FUNCTION_BLOCK Server_ALL (* Composite Function Block Type *)
  (* Standard: 61499-2 *)
  (* Version 0.0, 2018-11-07, 4DIAC-IDE, 4DIAC-Consortium *)
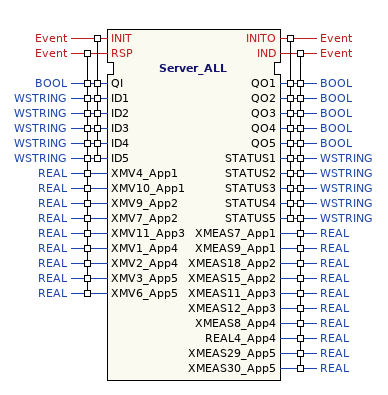
  EVENT_INPUT
    INIT WITH QI, ID1, ID2, ID4, ID5, ID3; (* Initialization Request *)
    RSP WITH QI, ID1, ID2, ID3, ID4, ID5, XMV4_App1, XMV10_App1, XMV9_App2, XMV7_App2, XMV11_App3, XMV1_App4, XMV2_App4, XMV3_App5, XMV6_App5; (* Normal Execution Request *)
  END_EVENT
  EVENT_OUTPUT
    INITO WITH QO1, QO3, QO2, QO4, QO5, STATUS1, STATUS2, STATUS3, STATUS4, STATUS5; (* Initialization Confirm *)
    IND WITH QO1, QO2, QO3, QO4, QO5, STATUS2, STATUS1, STATUS3, STATUS4, STATUS5, XMEAS7_App1, XMEAS9_App1, XMEAS18_App2, XMEAS15_App2, XMEAS11_App3, XMEAS12_App3, XMEAS8_App4, REAL4_App4, XMEAS29_App5, XMEAS30_App5; (* Execution Confirmation *)
  END_EVENT
  VAR_INPUT
    QI : BOOL; (* Input event qualifier *)
    ID1 : WSTRING;
    ID2 : WSTRING;
    ID3 : WSTRING;
    ID4 : WSTRING;
    ID5 : WSTRING;
    XMV4_App1 : REAL;
    XMV10_App1 : REAL;
    XMV9_App2 : REAL;
    XMV7_App2 : REAL;
    XMV11_App3 : REAL;
    XMV1_App4 : REAL;
    XMV2_App4 : REAL;
    XMV3_App5 : REAL;
    XMV6_App5 : REAL;
  END_VAR
  VAR_OUTPUT
    QO1 : BOOL; (* Output event qualifier *)
    QO2 : BOOL;
    QO3 : BOOL;
    QO4 : BOOL;
    QO5 : BOOL;
    STATUS1 : WSTRING;
    STATUS2 : WSTRING;
    STATUS3 : WSTRING;
    STATUS4 : WSTRING;
    STATUS5 : WSTRING;
    XMEAS7_App1 : REAL;
    XMEAS9_App1 : REAL;
    XMEAS18_App2 : REAL;
    XMEAS15_App2 : REAL;
    XMEAS11_App3 : REAL;
    XMEAS12_App3 : REAL;
    XMEAS8_App4 : REAL;
    REAL4_App4 : REAL;
    XMEAS29_App5 : REAL;
    XMEAS30_App5 : REAL;
  END_VAR
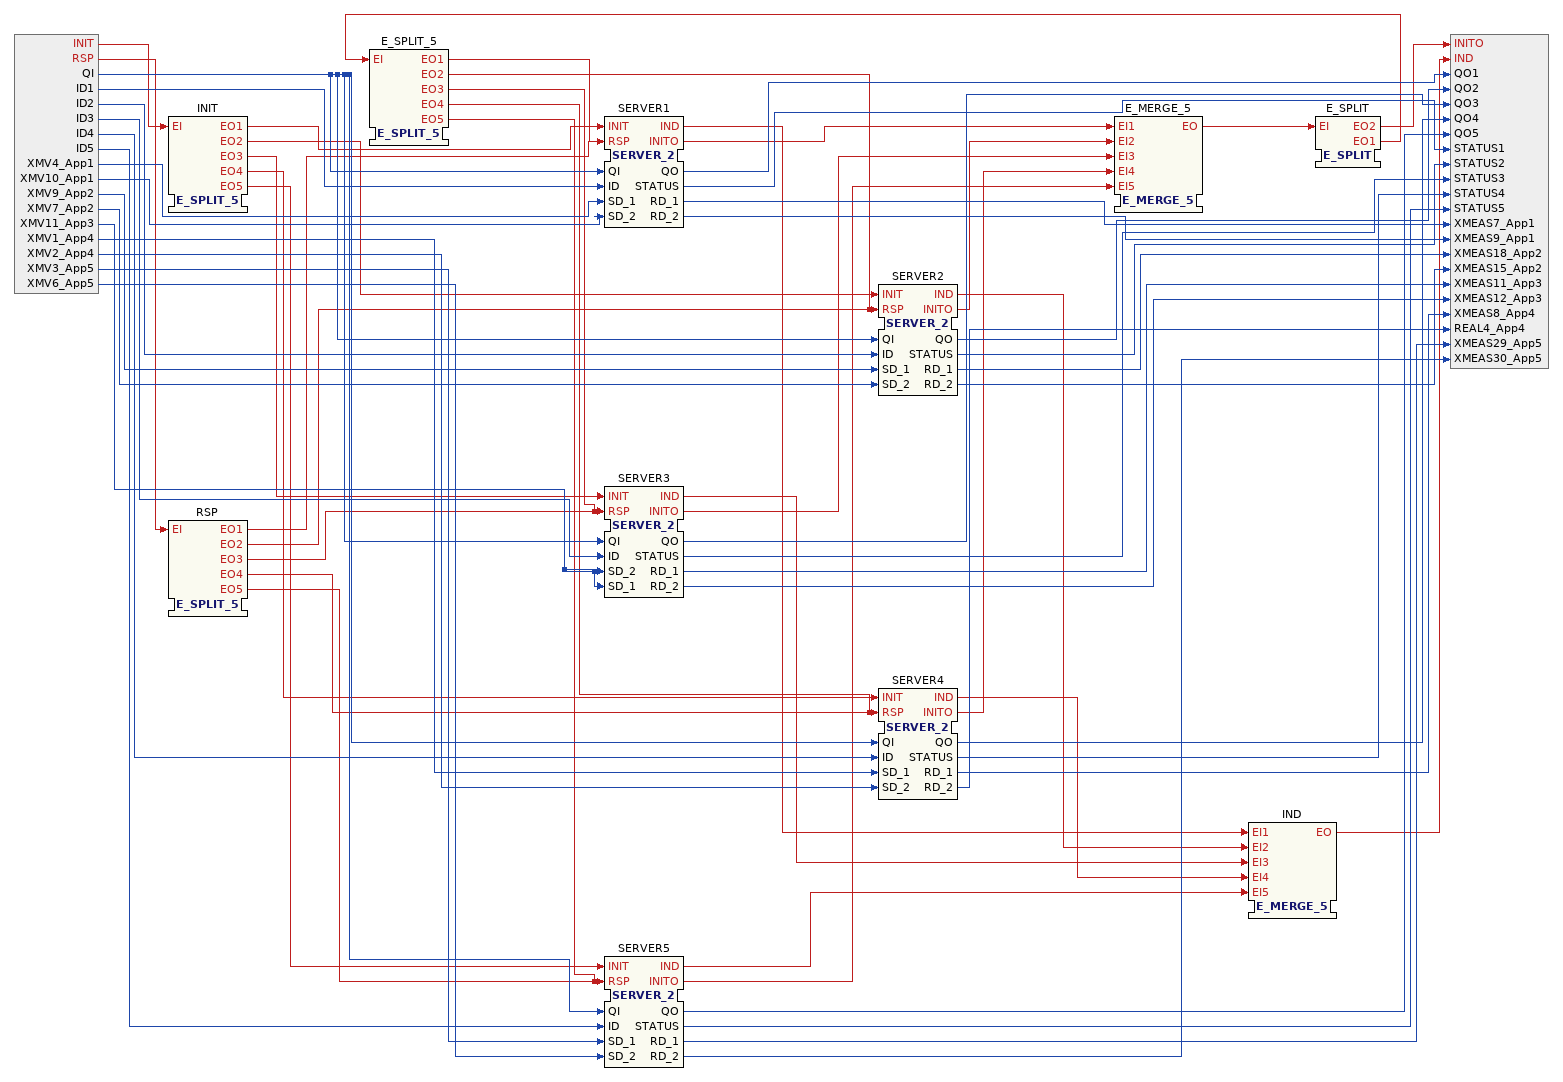
  FBS
    SERVER1 : SERVER_2;
    SERVER3 : SERVER_2;
    SERVER5 : SERVER_2;
    SERVER2 : SERVER_2;
    SERVER4 : SERVER_2;
    INIT : E_SPLIT_5;
    RSP : E_SPLIT_5;
    IND : E_MERGE_5;
    E_MERGE_5 : E_MERGE_5;
    E_SPLIT : E_SPLIT;
    E_SPLIT_5 : E_SPLIT_5;
  END_FBS
  EVENT_CONNECTIONS
    INIT.EO1 TO SERVER1.INIT;
    INIT.EO2 TO SERVER2.INIT;
    INIT.EO3 TO SERVER3.INIT;
    INIT.EO4 TO SERVER4.INIT;
    INIT.EO5 TO SERVER5.INIT;
    INIT TO INIT.EI;
    RSP TO RSP.EI;
    RSP.EO1 TO SERVER1.RSP;
    RSP.EO2 TO SERVER2.RSP;
    RSP.EO3 TO SERVER3.RSP;
    RSP.EO4 TO SERVER4.RSP;
    RSP.EO5 TO SERVER5.RSP;
    SERVER1.IND TO IND.EI1;
    SERVER2.IND TO IND.EI2;
    SERVER3.IND TO IND.EI3;
    SERVER4.IND TO IND.EI4;
    SERVER5.IND TO IND.EI5;
    IND.EO TO IND;
    SERVER1.INITO TO E_MERGE_5.EI1;
    SERVER2.INITO TO E_MERGE_5.EI2;
    SERVER3.INITO TO E_MERGE_5.EI3;
    SERVER4.INITO TO E_MERGE_5.EI4;
    SERVER5.INITO TO E_MERGE_5.EI5;
    E_MERGE_5.EO TO E_SPLIT.EI;
    E_SPLIT.EO2 TO INITO;
    E_SPLIT.EO1 TO E_SPLIT_5.EI;
    E_SPLIT_5.EO1 TO SERVER1.RSP;
    E_SPLIT_5.EO2 TO SERVER2.RSP;
    E_SPLIT_5.EO3 TO SERVER3.RSP;
    E_SPLIT_5.EO4 TO SERVER4.RSP;
    E_SPLIT_5.EO5 TO SERVER5.RSP;
  END_CONNECTIONS
  DATA_CONNECTIONS
    QI TO SERVER1.QI;
    QI TO SERVER2.QI;
    QI TO SERVER3.QI;
    QI TO SERVER4.QI;
    QI TO SERVER5.QI;
    ID1 TO SERVER1.ID;
    ID2 TO SERVER2.ID;
    ID3 TO SERVER3.ID;
    ID4 TO SERVER4.ID;
    ID5 TO SERVER5.ID;
    XMV4_App1 TO SERVER1.SD_1;
    XMV10_App1 TO SERVER1.SD_2;
    XMV9_App2 TO SERVER2.SD_1;
    XMV7_App2 TO SERVER2.SD_2;
    XMV11_App3 TO SERVER3.SD_2;
    XMV1_App4 TO SERVER4.SD_1;
    XMV2_App4 TO SERVER4.SD_2;
    XMV3_App5 TO SERVER5.SD_1;
    XMV6_App5 TO SERVER5.SD_2;
    SERVER1.QO TO QO1;
    SERVER2.QO TO QO2;
    SERVER3.QO TO QO3;
    SERVER4.QO TO QO4;
    SERVER5.QO TO QO5;
    SERVER1.STATUS TO STATUS1;
    SERVER2.STATUS TO STATUS2;
    SERVER3.STATUS TO STATUS3;
    SERVER4.STATUS TO STATUS4;
    SERVER5.STATUS TO STATUS5;
    SERVER1.RD_1 TO XMEAS7_App1;
    SERVER1.RD_2 TO XMEAS9_App1;
    SERVER2.RD_1 TO XMEAS18_App2;
    SERVER2.RD_2 TO XMEAS15_App2;
    SERVER3.RD_1 TO XMEAS11_App3;
    SERVER3.RD_2 TO XMEAS12_App3;
    SERVER4.RD_1 TO XMEAS8_App4;
    SERVER4.RD_2 TO REAL4_App4;
    SERVER5.RD_1 TO XMEAS29_App5;
    SERVER5.RD_2 TO XMEAS30_App5;
    XMV11_App3 TO SERVER3.SD_1;
  END_CONNECTIONS
END_FUNCTION_BLOCK
